Universal Robots PolyScope program: graub.urp

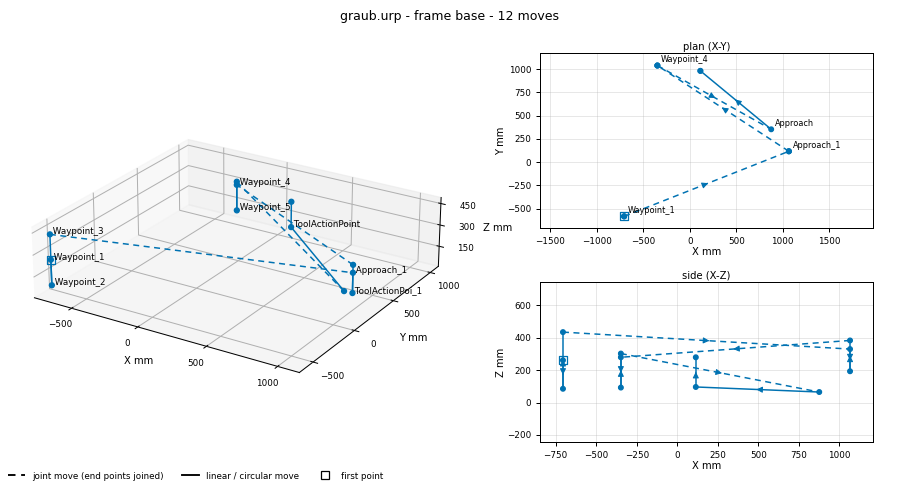
[picture p0: tool path of graub.urp in frame base, 12 of 12 moves have a stored position in this frame; points joined in program order, loops and branches not executed]
Program graub (installation=default directory=/home/ur/ursim-current/programs createdIn=5.8.0.10253 lastSavedIn=5.8.0.10253 robotSerialNumber=20195099999)
Calibrated DH parameters: a=[0, -0.6127, -0.57155, 0, 0, 0]; d=[0.1807, 0, 0, 0.17415, 0.11985, 0.11655]; alpha=[1.570796, 0, 0, 1.570796, -1.570796, 0]; deltaTheta=[0, 0, 0, 0, 0, 0]
Robot Program (runOnlyOnce=false)
  sensor := True
  MoveJ speed 60 deg/s, acceleration 80 deg/s^2 (useActiveTCP=true) feature=Base
    Waypoint Waypoint_1: TCP in base x=-705.224 y=-583.791 z=260.971 mm, rx=-0.0012 ry=3.1163 rz=0.0389 rad; joints [-129.442, -120.764, -93.953, -57.3, 90.2, -39.49] deg
    Wait Condition expression=sensor≟ True
  MoveL speed 250 mm/s, acceleration 1200 mm/s^2 (useActiveTCP=true) feature=Base
    Waypoint Waypoint_2: TCP in base x=-705.224 y=-583.791 z=84.929 mm, rx=-0.0012 ry=3.1163 rz=0.0389 rad; joints [-129.442, -131.824, -97.223, -42.971, 90.2, -39.49] deg
    Gripper := True
    Wait Sleep waitTime=1
    Waypoint Waypoint_3: TCP in base x=-705.224 y=-583.791 z=434.571 mm, rx=-0.0012 ry=3.1163 rz=0.0389 rad; joints [-129.442, -113.402, -85.773, -72.842, 90.2, -39.49] deg
    sensor := False
  URCap Palletizing (pallet-impl, Universal Robots) dataModel(palletFeature=Base, isPalletizing=true, Variable(key=name, variable(name=Pallet_1)), Variable(key=globalCountingVariable, variable(name=Pallet_1_cnt, initializeExpression=1)), Variable(key=layerNumberVariable, variable(name=Pallet_1_lno, initializeExpression=1)), Variable(key=layerCountingVariable, variable(name=Pallet_1_lct, initializeExpression=1)), Variable(key=handleSeparatorVariable, variable(name=Pallet_1_sep, initializeExpression=False)), Variable(key=totalCountVariable, variable(name=Pallet_1_tct, initializeExpression=1)), Variable(key=referencePoint, variable(featureName=referencePoint)), Variable(key=separatorPoint, variable(featureName=separatorPoint)), Length(key=objectHeight value=0.1 unit=M)); state(isChildrenLocked=true)
    URCap Patterns (pallet-impl, Universal Robots) dataModel(separator=true, Length(key=separatorHeight value=0.006 unit=M)); state(isChildrenLocked=true)
      URCap Pattern (pallet-impl, Universal Robots) dataModel(UUID=1b8fb367-97a9-435e-ad25-830c0d7c81cb, patternType=IRREGULAR, Variable(key=nameVariable, variable(name=Irreg_Pattern_1))); state(isChildrenLocked=true)
        URCap Item (pallet-impl, Universal Robots) dataModel(UUID=1b49ad4d-770f-44cd-9acf-c4c4b920f22e, patternType=IRREGULAR, index=0, calibrationDeltaTheta=[0.0, 0.0, 0.0, 0.0, 0.0, 0.0], calibrationA=[0.0, -0.6127, -0.57155, 0.0, 0.0, 0.0], calibrationD=[0.1807, 0.0, 0.0, 0.17415, 0.11985, 0.11655], calibrationAlpha=[1.570796327, 0.0, 0.0, 1.570796327, -1.570796327, 0.0], calibrationJointChecksum=[-1, -1, -1, -1, -1, -1], calibrationStatus=0, calibrationValidChecksum=false, baseToFeature=[0.0, 0.0, 0.0, 0.0, 0.0, 0.0], TCPOffset=[0.0, -1.3877787807814457E-17, 4.163336342344337E-16, 0.0, 0.0, 0.0], Variable(key=variable, variable(name=Item_1)), JointPositions(key=jointpositions, JointPosition(key=[1], Angle(key=pos value=0.271485 unit=RAD)), JointPosition(key=[2], Angle(key=pos value=-2.623067 unit=RAD)), JointPosition(key=[3], Angle(key=pos value=-1.299161 unit=RAD)), JointPosition(key=[4], Angle(key=pos value=-0.790161 unit=RAD)), JointPosition(key=[5], Angle(key=pos value=1.570796 unit=RAD)), JointPosition(key=[6], Angle(key=pos value=1.843513 unit=RAD))))
        URCap Item (pallet-impl, Universal Robots) dataModel(UUID=e09fed2d-4457-46ad-8b72-bf1af07cccc8, patternType=IRREGULAR, index=1, calibrationDeltaTheta=[0.0, 0.0, 0.0, 0.0, 0.0, 0.0], calibrationA=[0.0, -0.6127, -0.57155, 0.0, 0.0, 0.0], calibrationD=[0.1807, 0.0, 0.0, 0.17415, 0.11985, 0.11655], calibrationAlpha=[1.570796327, 0.0, 0.0, 1.570796327, -1.570796327, 0.0], calibrationJointChecksum=[-1, -1, -1, -1, -1, -1], calibrationStatus=0, calibrationValidChecksum=false, baseToFeature=[0.0, 0.0, 0.0, 0.0, 0.0, 0.0], TCPOffset=[2.220446049250313E-16, -3.469446951953614E-18, 4.440892098500626E-16, 0.0, 0.0, 0.0], Variable(key=variable, variable(name=Item_2)), JointPositions(key=jointpositions, JointPosition(key=[1], Angle(key=pos value=0.141494 unit=RAD)), JointPosition(key=[2], Angle(key=pos value=-2.667014 unit=RAD)), JointPosition(key=[3], Angle(key=pos value=-1.225905 unit=RAD)), JointPosition(key=[4], Angle(key=pos value=-0.81947 unit=RAD)), JointPosition(key=[5], Angle(key=pos value=1.570796 unit=RAD)), JointPosition(key=[6], Angle(key=pos value=1.713522 unit=RAD))))
        URCap Item (pallet-impl, Universal Robots) dataModel(UUID=7b299bc4-ada8-49d9-a477-8758a9ddf272, patternType=IRREGULAR, index=2, calibrationDeltaTheta=[0.0, 0.0, 0.0, 0.0, 0.0, 0.0], calibrationA=[0.0, -0.6127, -0.57155, 0.0, 0.0, 0.0], calibrationD=[0.1807, 0.0, 0.0, 0.17415, 0.11985, 0.11655], calibrationAlpha=[1.570796327, 0.0, 0.0, 1.570796327, -1.570796327, 0.0], calibrationJointChecksum=[-1, -1, -1, -1, -1, -1], calibrationStatus=0, calibrationValidChecksum=false, baseToFeature=[0.0, 0.0, 0.0, 0.0, 0.0, 0.0], TCPOffset=[2.220446049250313E-16, -4.163336342344337E-17, 1.8041124150158794E-16, 0.0, 0.0, 0.0], Variable(key=variable, variable(name=Item_3)), JointPositions(key=jointpositions, JointPosition(key=[1], Angle(key=pos value=0.128812 unit=RAD)), JointPosition(key=[2], Angle(key=pos value=-2.34045 unit=RAD)), JointPosition(key=[3], Angle(key=pos value=-2.091835 unit=RAD)), JointPosition(key=[4], Angle(key=pos value=-0.280103 unit=RAD)), JointPosition(key=[5], Angle(key=pos value=1.570796 unit=RAD)), JointPosition(key=[6], Angle(key=pos value=1.700841 unit=RAD))))
        URCap Item (pallet-impl, Universal Robots) dataModel(UUID=20383d34-7355-4a22-bc34-7da397a0ffe1, patternType=IRREGULAR, index=3, calibrationDeltaTheta=[0.0, 0.0, 0.0, 0.0, 0.0, 0.0], calibrationA=[0.0, -0.6127, -0.57155, 0.0, 0.0, 0.0], calibrationD=[0.1807, 0.0, 0.0, 0.17415, 0.11985, 0.11655], calibrationAlpha=[1.570796327, 0.0, 0.0, 1.570796327, -1.570796327, 0.0], calibrationJointChecksum=[-1, -1, -1, -1, -1, -1], calibrationStatus=0, calibrationValidChecksum=false, baseToFeature=[0.0, 0.0, 0.0, 0.0, 0.0, 0.0], TCPOffset=[1.1102230246251565E-16, -8.326672684688674E-17, 4.579669976578771E-16, 0.0, 0.0, 0.0], Variable(key=variable, variable(name=Item_4)), JointPositions(key=jointpositions, JointPosition(key=[1], Angle(key=pos value=0.401415 unit=RAD)), JointPosition(key=[2], Angle(key=pos value=-2.396838 unit=RAD)), JointPosition(key=[3], Angle(key=pos value=-2.012159 unit=RAD)), JointPosition(key=[4], Angle(key=pos value=-0.303392 unit=RAD)), JointPosition(key=[5], Angle(key=pos value=1.570796 unit=RAD)), JointPosition(key=[6], Angle(key=pos value=1.973443 unit=RAD))))
      URCap Pattern (pallet-impl, Universal Robots) dataModel(UUID=08873cfb-372a-4e66-ad47-c7f4bdadf5b3, patternType=IRREGULAR, columns=3, rows=4, objects=3, Variable(key=nameVariable, variable(name=Irreg_Pattern_2))); state(isChildrenLocked=true)
        URCap Item (pallet-impl, Universal Robots) dataModel(UUID=622b5cf1-2ea0-4e82-a6c7-17ae4498ee9b, patternType=IRREGULAR, index=0, calibrationDeltaTheta=[0.0, 0.0, 0.0, 0.0, 0.0, 0.0], calibrationA=[0.0, -0.6127, -0.57155, 0.0, 0.0, 0.0], calibrationD=[0.1807, 0.0, 0.0, 0.17415, 0.11985, 0.11655], calibrationAlpha=[1.570796327, 0.0, 0.0, 1.570796327, -1.570796327, 0.0], calibrationJointChecksum=[-1, -1, -1, -1, -1, -1], calibrationStatus=0, calibrationValidChecksum=false, baseToFeature=[0.0, 0.0, 0.0, 0.0, 0.0, 0.0], TCPOffset=[2.220446049250313E-16, -9.71445146547012E-17, 2.7755575615628914E-16, 0.0, 0.0, 0.0], Variable(key=variable, variable(name=Item_5)), JointPositions(key=jointpositions, JointPosition(key=[1], Angle(key=pos value=0.271485 unit=RAD)), JointPosition(key=[2], Angle(key=pos value=-2.381996 unit=RAD)), JointPosition(key=[3], Angle(key=pos value=-1.286774 unit=RAD)), JointPosition(key=[4], Angle(key=pos value=-1.043619 unit=RAD)), JointPosition(key=[5], Angle(key=pos value=1.570796 unit=RAD)), JointPosition(key=[6], Angle(key=pos value=1.843513 unit=RAD))))
        URCap Item (pallet-impl, Universal Robots) dataModel(UUID=1d731585-ca26-4218-9cac-7a63b7a7439d, patternType=IRREGULAR, index=1, calibrationDeltaTheta=[0.0, 0.0, 0.0, 0.0, 0.0, 0.0], calibrationA=[0.0, -0.6127, -0.57155, 0.0, 0.0, 0.0], calibrationD=[0.1807, 0.0, 0.0, 0.17415, 0.11985, 0.11655], calibrationAlpha=[1.570796327, 0.0, 0.0, 1.570796327, -1.570796327, 0.0], calibrationJointChecksum=[-1, -1, -1, -1, -1, -1], calibrationStatus=0, calibrationValidChecksum=false, baseToFeature=[0.0, 0.0, 0.0, 0.0, 0.0, 0.0], TCPOffset=[0.0, -1.3877787807814457E-17, 4.996003610813204E-16, 0.0, 0.0, 0.0], Variable(key=variable, variable(name=Item_6)), JointPositions(key=jointpositions, JointPosition(key=[1], Angle(key=pos value=0.141494 unit=RAD)), JointPosition(key=[2], Angle(key=pos value=-2.428419 unit=RAD)), JointPosition(key=[3], Angle(key=pos value=-1.22148 unit=RAD)), JointPosition(key=[4], Angle(key=pos value=-1.06249 unit=RAD)), JointPosition(key=[5], Angle(key=pos value=1.570796 unit=RAD)), JointPosition(key=[6], Angle(key=pos value=1.713522 unit=RAD))))
        URCap Item (pallet-impl, Universal Robots) dataModel(UUID=2db7b465-85fe-4914-b818-ef91deeb26bb, patternType=IRREGULAR, index=2, calibrationDeltaTheta=[0.0, 0.0, 0.0, 0.0, 0.0, 0.0], calibrationA=[0.0, -0.6127, -0.57155, 0.0, 0.0, 0.0], calibrationD=[0.1807, 0.0, 0.0, 0.17415, 0.11985, 0.11655], calibrationAlpha=[1.570796327, 0.0, 0.0, 1.570796327, -1.570796327, 0.0], calibrationJointChecksum=[-1, -1, -1, -1, -1, -1], calibrationStatus=0, calibrationValidChecksum=false, baseToFeature=[0.0, 0.0, 0.0, 0.0, 0.0, 0.0], TCPOffset=[2.220446049250313E-16, -2.7755575615628914E-17, 2.7755575615628914E-16, 0.0, 0.0, 0.0], Variable(key=variable, variable(name=Item_7)), JointPositions(key=jointpositions, JointPosition(key=[1], Angle(key=pos value=0.128812 unit=RAD)), JointPosition(key=[2], Angle(key=pos value=-2.023197 unit=RAD)), JointPosition(key=[3], Angle(key=pos value=-2.102216 unit=RAD)), JointPosition(key=[4], Angle(key=pos value=-0.586976 unit=RAD)), JointPosition(key=[5], Angle(key=pos value=1.570796 unit=RAD)), JointPosition(key=[6], Angle(key=pos value=1.700841 unit=RAD))))
        URCap Item (pallet-impl, Universal Robots) dataModel(UUID=a88a78f6-847e-422b-a6a2-fda344ad4760, patternType=IRREGULAR, index=3, calibrationDeltaTheta=[0.0, 0.0, 0.0, 0.0, 0.0, 0.0], calibrationA=[0.0, -0.6127, -0.57155, 0.0, 0.0, 0.0], calibrationD=[0.1807, 0.0, 0.0, 0.17415, 0.11985, 0.11655], calibrationAlpha=[1.570796327, 0.0, 0.0, 1.570796327, -1.570796327, 0.0], calibrationJointChecksum=[-1, -1, -1, -1, -1, -1], calibrationStatus=0, calibrationValidChecksum=false, baseToFeature=[0.0, 0.0, 0.0, 0.0, 0.0, 0.0], TCPOffset=[1.1102230246251565E-16, -2.7755575615628914E-17, 3.3306690738754696E-16, 0.0, 0.0, 0.0], Variable(key=variable, variable(name=Item_8)), JointPositions(key=jointpositions, JointPosition(key=[1], Angle(key=pos value=0.401415 unit=RAD)), JointPosition(key=[2], Angle(key=pos value=-2.004712 unit=RAD)), JointPosition(key=[3], Angle(key=pos value=-2.018046 unit=RAD)), JointPosition(key=[4], Angle(key=pos value=-0.689631 unit=RAD)), JointPosition(key=[5], Angle(key=pos value=1.570796 unit=RAD)), JointPosition(key=[6], Angle(key=pos value=1.973443 unit=RAD))))
      URCap Pattern (pallet-impl, Universal Robots) dataModel(UUID=aee68c81-00e4-4400-9c79-0f60ee43e765, patternType=IRREGULAR, columns=3, rows=4, objects=3, Variable(key=nameVariable, variable(name=Irreg_Pattern_3))); state(isChildrenLocked=true)
        URCap Item (pallet-impl, Universal Robots) dataModel(UUID=d2103d47-dda9-4b36-a16c-b2c0b133670e, patternType=IRREGULAR, index=0, calibrationDeltaTheta=[0.0, 0.0, 0.0, 0.0, 0.0, 0.0], calibrationA=[0.0, -0.6127, -0.57155, 0.0, 0.0, 0.0], calibrationD=[0.1807, 0.0, 0.0, 0.17415, 0.11985, 0.11655], calibrationAlpha=[1.570796327, 0.0, 0.0, 1.570796327, -1.570796327, 0.0], calibrationJointChecksum=[-1, -1, -1, -1, -1, -1], calibrationStatus=0, calibrationValidChecksum=false, baseToFeature=[0.0, 0.0, 0.0, 0.0, 0.0, 0.0], TCPOffset=[-2.220446049250313E-16, 5.551115123125783E-17, 5.551115123125783E-16, 0.0, 0.0, 0.0], Variable(key=variable, variable(name=Item_9)), JointPositions(key=jointpositions, JointPosition(key=[1], Angle(key=pos value=0.271485 unit=RAD)), JointPosition(key=[2], Angle(key=pos value=-2.234405 unit=RAD)), JointPosition(key=[3], Angle(key=pos value=-1.101196 unit=RAD)), JointPosition(key=[4], Angle(key=pos value=-1.376789 unit=RAD)), JointPosition(key=[5], Angle(key=pos value=1.570796 unit=RAD)), JointPosition(key=[6], Angle(key=pos value=1.843513 unit=RAD))))
        URCap Item (pallet-impl, Universal Robots) dataModel(UUID=f2ce0ae9-3a10-43a1-a5d6-39bc4666baa3, patternType=IRREGULAR, index=1, calibrationDeltaTheta=[0.0, 0.0, 0.0, 0.0, 0.0, 0.0], calibrationA=[0.0, -0.6127, -0.57155, 0.0, 0.0, 0.0], calibrationD=[0.1807, 0.0, 0.0, 0.17415, 0.11985, 0.11655], calibrationAlpha=[1.570796327, 0.0, 0.0, 1.570796327, -1.570796327, 0.0], calibrationJointChecksum=[-1, -1, -1, -1, -1, -1], calibrationStatus=0, calibrationValidChecksum=false, baseToFeature=[0.0, 0.0, 0.0, 0.0, 0.0, 0.0], TCPOffset=[0.0, -1.0408340855860843E-17, 4.996003610813204E-16, 0.0, 0.0, 0.0], Variable(key=variable, variable(name=Item_10)), JointPositions(key=jointpositions, JointPosition(key=[1], Angle(key=pos value=0.141494 unit=RAD)), JointPosition(key=[2], Angle(key=pos value=-2.287321 unit=RAD)), JointPosition(key=[3], Angle(key=pos value=-1.053312 unit=RAD)), JointPosition(key=[4], Angle(key=pos value=-1.371757 unit=RAD)), JointPosition(key=[5], Angle(key=pos value=1.570796 unit=RAD)), JointPosition(key=[6], Angle(key=pos value=1.713522 unit=RAD))))
        URCap Item (pallet-impl, Universal Robots) dataModel(UUID=dc30364b-b3d3-4c02-947e-90c0441e133f, patternType=IRREGULAR, index=2, calibrationDeltaTheta=[0.0, 0.0, 0.0, 0.0, 0.0, 0.0], calibrationA=[0.0, -0.6127, -0.57155, 0.0, 0.0, 0.0], calibrationD=[0.1807, 0.0, 0.0, 0.17415, 0.11985, 0.11655], calibrationAlpha=[1.570796327, 0.0, 0.0, 1.570796327, -1.570796327, 0.0], calibrationJointChecksum=[-1, -1, -1, -1, -1, -1], calibrationStatus=0, calibrationValidChecksum=false, baseToFeature=[0.0, 0.0, 0.0, 0.0, 0.0, 0.0], TCPOffset=[1.1102230246251565E-16, -4.163336342344337E-17, 2.7755575615628914E-16, 0.0, 0.0, 0.0], Variable(key=variable, variable(name=Item_11)), JointPositions(key=jointpositions, JointPosition(key=[1], Angle(key=pos value=0.128812 unit=RAD)), JointPosition(key=[2], Angle(key=pos value=-1.66209 unit=RAD)), JointPosition(key=[3], Angle(key=pos value=-1.870019 unit=RAD)), JointPosition(key=[4], Angle(key=pos value=-1.18028 unit=RAD)), JointPosition(key=[5], Angle(key=pos value=1.570796 unit=RAD)), JointPosition(key=[6], Angle(key=pos value=1.700841 unit=RAD))))
        URCap Item (pallet-impl, Universal Robots) dataModel(UUID=6d17dbee-1df2-4bbf-8e81-30d1b7cdde83, patternType=IRREGULAR, index=3, calibrationDeltaTheta=[0.0, 0.0, 0.0, 0.0, 0.0, 0.0], calibrationA=[0.0, -0.6127, -0.57155, 0.0, 0.0, 0.0], calibrationD=[0.1807, 0.0, 0.0, 0.17415, 0.11985, 0.11655], calibrationAlpha=[1.570796327, 0.0, 0.0, 1.570796327, -1.570796327, 0.0], calibrationJointChecksum=[-1, -1, -1, -1, -1, -1], calibrationStatus=0, calibrationValidChecksum=false, baseToFeature=[0.0, 0.0, 0.0, 0.0, 0.0, 0.0], TCPOffset=[2.220446049250313E-16, -1.6653345369377348E-16, 2.7755575615628914E-16, 0.0, 0.0, 0.0], Variable(key=variable, variable(name=Item_12)), JointPositions(key=jointpositions, JointPosition(key=[1], Angle(key=pos value=0.401415 unit=RAD)), JointPosition(key=[2], Angle(key=pos value=-1.696005 unit=RAD)), JointPosition(key=[3], Angle(key=pos value=-1.753143 unit=RAD)), JointPosition(key=[4], Angle(key=pos value=-1.263242 unit=RAD)), JointPosition(key=[5], Angle(key=pos value=1.570796 unit=RAD)), JointPosition(key=[6], Angle(key=pos value=1.973443 unit=RAD))))
      URCap Item (pallet-impl, Universal Robots) dataModel(UUID=691122ae-95dd-404c-816a-a51f7764fe50, patternType=SEPARATOR, index=0, calibrationDeltaTheta=[0.0, 0.0, 0.0, 0.0, 0.0, 0.0], calibrationA=[0.0, -0.6127, -0.57155, 0.0, 0.0, 0.0], calibrationD=[0.1807, 0.0, 0.0, 0.17415, 0.11985, 0.11655], calibrationAlpha=[1.570796327, 0.0, 0.0, 1.570796327, -1.570796327, 0.0], calibrationJointChecksum=[-1, -1, -1, -1, -1, -1], calibrationStatus=0, calibrationValidChecksum=false, baseToFeature=[0.0, 0.0, 0.0, 0.0, 0.0, 0.0], TCPOffset=[-1.3877787807814457E-17, -2.220446049250313E-16, 3.608224830031759E-16, 0.0, 0.0, 0.0], Variable(key=variable, variable(name=Separator)), JointPositions(key=jointpositions, JointPosition(key=[1], Angle(key=pos value=1.631889 unit=RAD)), JointPosition(key=[2], Angle(key=pos value=-2.370296 unit=RAD)), JointPosition(key=[3], Angle(key=pos value=-1.534688 unit=RAD)), JointPosition(key=[4], Angle(key=pos value=-0.807405 unit=RAD)), JointPosition(key=[5], Angle(key=pos value=1.570796 unit=RAD)), JointPosition(key=[6], Angle(key=pos value=3.203917 unit=RAD))))
    URCap Layers (pallet-impl, Universal Robots) dataModel(selectedPatterns=[1b8fb367-97a9-435e-ad25-830c0d7c81cb, 08873cfb-372a-4e66-ad47-c7f4bdadf5b3, aee68c81-00e4-4400-9c79-0f60ee43e765, 1b8fb367-97a9-435e-ad25-830c0d7c81cb], separators=[true, true, true, false])
    URCap At Each Item (pallet-impl, Universal Robots) dataModel(selectedPattern=1b8fb367-97a9-435e-ad25-830c0d7c81cb, selectedPosition=1b49ad4d-770f-44cd-9acf-c4c4b920f22e, Approach_calibrationDeltaTheta=[0.0, 0.0, 0.0, 0.0, 0.0, 0.0], Approach_calibrationA=[0.0, -0.6127, -0.57155, 0.0, 0.0, 0.0], Approach_calibrationD=[0.1807, 0.0, 0.0, 0.17415, 0.11985, 0.11655], Approach_calibrationAlpha=[1.570796327, 0.0, 0.0, 1.570796327, -1.570796327, 0.0], Approach_calibrationJointChecksum=[-1, -1, -1, -1, -1, -1], Approach_calibrationStatus=0, Approach_calibrationValidChecksum=false, Approach_baseToFeature=[0.0, 0.0, 0.0, 0.0, 0.0, 0.0], Approach_TCPOffset=[0.0, -2.7755575615628914E-17, 4.440892098500626E-16, 0.0, 0.0, 0.0], Exit_calibrationDeltaTheta=[0.0, 0.0, 0.0, 0.0, 0.0, 0.0], Exit_calibrationA=[0.0, -0.6127, -0.57155, 0.0, 0.0, 0.0], Exit_calibrationD=[0.1807, 0.0, 0.0, 0.17415, 0.11985, 0.11655], Exit_calibrationAlpha=[1.570796327, 0.0, 0.0, 1.570796327, -1.570796327, 0.0], Exit_calibrationJointChecksum=[-1, -1, -1, -1, -1, -1], Exit_calibrationStatus=0, Exit_calibrationValidChecksum=false, Exit_baseToFeature=[0.0, 0.0, 0.0, 0.0, 0.0, 0.0], Exit_TCPOffset=[0.0, -1.3877787807814457E-17, 3.885780586188048E-16, 0.0, 0.0, 0.0], currentWizardState=LANDING, Pose(key=refBaseToFeature, Position(key=posePosition, Length(key=X value=0 unit=M), Length(key=Y value=0 unit=M), Length(key=Z value=0 unit=M)), Rotation(key=poseRotation, Angle(key=RX value=0 unit=RAD), Angle(key=RY value=0 unit=RAD), Angle(key=RZ value=0 unit=RAD))), Pose(key=refPose, Position(key=posePosition, Length(key=X value=1.066025 unit=M), Length(key=Y value=0.115965 unit=M), Length(key=Z value=0.193029 unit=M)), Rotation(key=poseRotation, Angle(key=RX value=0.001935 unit=RAD), Angle(key=RY value=3.141592 unit=RAD), Angle(key=RZ value=0 unit=RAD))), JointPositions(key=Approach_jointpositions, JointPosition(key=[1], Angle(key=pos value=0.271485 unit=RAD)), JointPosition(key=[2], Angle(key=pos value=-2.285759 unit=RAD)), JointPosition(key=[3], Angle(key=pos value=-1.207615 unit=RAD)), JointPosition(key=[4], Angle(key=pos value=-1.219015 unit=RAD)), JointPosition(key=[5], Angle(key=pos value=1.570796 unit=RAD)), JointPosition(key=[6], Angle(key=pos value=1.843513 unit=RAD))), JointPositions(key=Exit_jointpositions, JointPosition(key=[1], Angle(key=pos value=0.271485 unit=RAD)), JointPosition(key=[2], Angle(key=pos value=-2.256854 unit=RAD)), JointPosition(key=[3], Angle(key=pos value=-1.159651 unit=RAD)), JointPosition(key=[4], Angle(key=pos value=-1.295883 unit=RAD)), JointPosition(key=[5], Angle(key=pos value=1.570796 unit=RAD)), JointPosition(key=[6], Angle(key=pos value=1.843513 unit=RAD))))
      URCap Generated Movements (pallet-impl, Universal Robots) state(isChildrenLocked=true)
        MoveJ speed 60 deg/s, acceleration 80 deg/s^2 (useActiveTCP=true) feature=referencePoint
          Waypoint Approach_1: TCP in base x=1066.025 y=115.965 z=329.871 mm, rx=0.0019 ry=3.1416 rz=0 rad; joints [15.555, -130.964, -69.191, -69.844, 90, 105.626] deg; TCP offset x=0 y=0 z=0 mm, rx=0 ry=0 rz=0 rad; feature pose in base x=1066.025 y=115.965 z=193.029 mm, rx=0.0019 ry=3.1416 rz=0 rad
        MoveL speed 250 mm/s, acceleration 1200 mm/s^2 (useActiveTCP=true) feature(featureName=referencePoint)
          Waypoint ToolActionPoi_1: TCP in base x=1066.025 y=115.965 z=193.029 mm, rx=0.0019 ry=3.1416 rz=0 rad; joints [15.555, -136.749, -73.85, -59.401, 90, 105.626] deg; TCP offset x=0 y=0 z=0 mm, rx=0 ry=0 rz=0 rad
        Folder Tool action
          Gripper := False
          Wait Sleep waitTime=1
        MoveL speed 250 mm/s, acceleration 1200 mm/s^2 (useActiveTCP=true) feature(featureName=referencePoint)
          Waypoint Exit_2: TCP in base x=1066.025 y=115.965 z=383.071 mm, rx=0.0019 ry=3.1416 rz=0 rad; joints [15.555, -129.308, -66.443, -74.249, 90, 105.626] deg; TCP offset x=0 y=0 z=0 mm, rx=0 ry=0 rz=0 rad
    URCap Separator Action (pallet-impl, Universal Robots) dataModel(Approach_calibrationDeltaTheta=[0.0, 0.0, 0.0, 0.0, 0.0, 0.0], Approach_calibrationA=[0.0, -0.6127, -0.57155, 0.0, 0.0, 0.0], Approach_calibrationD=[0.1807, 0.0, 0.0, 0.17415, 0.11985, 0.11655], Approach_calibrationAlpha=[1.570796327, 0.0, 0.0, 1.570796327, -1.570796327, 0.0], Approach_calibrationJointChecksum=[-1, -1, -1, -1, -1, -1], Approach_calibrationStatus=0, Approach_calibrationValidChecksum=false, Approach_baseToFeature=[0.0, 0.0, 0.0, 0.0, 0.0, 0.0], Approach_TCPOffset=[3.3306690738754696E-16, -1.1102230246251565E-16, 4.0245584642661925E-16, 0.0, 0.0, 0.0], Exit_calibrationDeltaTheta=[0.0, 0.0, 0.0, 0.0, 0.0, 0.0], Exit_calibrationA=[0.0, -0.6127, -0.57155, 0.0, 0.0, 0.0], Exit_calibrationD=[0.1807, 0.0, 0.0, 0.17415, 0.11985, 0.11655], Exit_calibrationAlpha=[1.570796327, 0.0, 0.0, 1.570796327, -1.570796327, 0.0], Exit_calibrationJointChecksum=[-1, -1, -1, -1, -1, -1], Exit_calibrationStatus=0, Exit_calibrationValidChecksum=false, Exit_baseToFeature=[0.0, 0.0, 0.0, 0.0, 0.0, 0.0], Exit_TCPOffset=[0.0, -2.220446049250313E-16, 3.885780586188048E-16, 0.0, 0.0, 0.0], currentWizardState=LANDING, JointPositions(key=Approach_jointpositions, JointPosition(key=[1], Angle(key=pos value=0.567861 unit=RAD)), JointPosition(key=[2], Angle(key=pos value=-2.357547 unit=RAD)), JointPosition(key=[3], Angle(key=pos value=-1.64073 unit=RAD)), JointPosition(key=[4], Angle(key=pos value=-0.714112 unit=RAD)), JointPosition(key=[5], Angle(key=pos value=1.570796 unit=RAD)), JointPosition(key=[6], Angle(key=pos value=2.139889 unit=RAD))), JointPositions(key=Exit_jointpositions, JointPosition(key=[1], Angle(key=pos value=1.631889 unit=RAD)), JointPosition(key=[2], Angle(key=pos value=-2.19074 unit=RAD)), JointPosition(key=[3], Angle(key=pos value=-1.469871 unit=RAD)), JointPosition(key=[4], Angle(key=pos value=-1.051778 unit=RAD)), JointPosition(key=[5], Angle(key=pos value=1.570796 unit=RAD)), JointPosition(key=[6], Angle(key=pos value=3.203917 unit=RAD))))
      Folder Pick Up Separator
        MoveJ speed 60 deg/s, acceleration 80 deg/s^2 (useActiveTCP=true) feature=Base
          Waypoint Waypoint_4: TCP in base x=-347.941 y=1038.15 z=279.329 mm, rx=0.0019 ry=3.1416 rz=0 rad; joints [117.681, -134.959, -67.504, -67.537, 90, 207.751] deg
        MoveL speed 250 mm/s, acceleration 1200 mm/s^2 (useActiveTCP=true) feature=Base
          Waypoint Waypoint_5: TCP in base x=-347.941 y=1038.15 z=92.344 mm, rx=0.0019 ry=3.1416 rz=0 rad; joints [117.681, -144.012, -71.479, -54.508, 90, 207.751] deg
          Gripper := True
          Wait Sleep waitTime=1
          Waypoint Waypoint_6: TCP in base x=-347.941 y=1038.15 z=302.286 mm, rx=0.0019 ry=3.1416 rz=0 rad; joints [117.681, -134.101, -66.579, -69.319, 90, 207.751] deg
      MoveJ speed 60 deg/s, acceleration 80 deg/s^2 (useActiveTCP=true) feature=separatorPoint
        Waypoint Approach: TCP in base x=876.029 y=352.296 z=64.902 mm, rx=0.0019 ry=3.1416 rz=0 rad; joints [32.536, -135.078, -94.007, -40.916, 90, 122.607] deg; TCP offset x=0 y=0 z=0 mm, rx=0 ry=0 rz=0 rad; feature pose in base x=114.473 y=980.922 z=96.086 mm, rx=0.0019 ry=3.1416 rz=0 rad
      MoveL speed 250 mm/s, acceleration 1200 mm/s^2 (useActiveTCP=true) feature(featureName=separatorPoint)
        Waypoint ToolActionPoint: TCP in base x=114.473 y=980.922 z=96.086 mm, rx=0.0019 ry=3.1416 rz=0 rad; joints [93.5, -135.808, -87.931, -46.261, 90, 183.571] deg; TCP offset x=0 y=0 z=0 mm, rx=0 ry=0 rz=0 rad
      Folder Tool action
        Gripper := False
        Wait Sleep waitTime=1
      MoveL speed 250 mm/s, acceleration 1200 mm/s^2 (useActiveTCP=true) feature(featureName=separatorPoint)
        Waypoint Exit_1: TCP in base x=114.473 y=980.922 z=279.329 mm, rx=0.0019 ry=3.1416 rz=0 rad; joints [93.5, -125.52, -84.217, -60.262, 90, 183.571] deg; TCP offset x=0 y=0 z=0 mm, rx=0 ry=0 rz=0 rad
